// TIA Portal V16 export
// export: Created 2023-08-28T09:37:51.4907013Z, ExportSetting WithDefaults, DisplayName Totally Integrated Automation Portal, DisplayVersion V16 Update 6, DisplayName TIA Portal Version Control Interface, DisplayVersion V16 Update 2, DisplayName TIA Portal Openness, DisplayVersion V16 Update 6, DisplayName STEP 7 Professional, DisplayVersion V16 Update 6, DisplayName STEP 7 Safety, DisplayVersion V16, DisplayName WinCC Advanced, DisplayVersion V16 Update 6
DATA_BLOCK "dbModbusRTU_Reg"   // DB37
TITLE = Modbus RTU Data
{ S7_Optimized_Access := 'FALSE' }
AUTHOR : RTecmer
VERSION : 0.1
// Dane pomiarowe przekazane z bloku danych master modbus RTU
// stored: AutoNumber true, DBAccessibleFromOPCUA true, IsOnlyStoredInLoadMemory false, IsWriteProtectedInAS false
   VAR
      received_6_Wielkość_przeływu_Adres_0 { S7_SetPoint := 'True'} : "typeDataABB_DWord";   // wielkość przepływu
      received_6_Licznik_objętość_VF_Adres_2 { S7_SetPoint := 'True'} : "typeDataABB_DWord";   // licznik objętości VF
      received_6_Licznik_objętość_VR_Adres_4 { S7_SetPoint := 'True'} : "typeDataABB_DWord";   // licznik objętości VR
      received_6_Licznik_różnicowy_VD_Adres_6 { S7_SetPoint := 'True'} : "typeDataABB_DWord";   // licznik różnicy
      receive_6_Stan_licz_bjętości_GF_Adres_8 { S7_SetPoint := 'True'} : "typeDataABB_DWord";   // licznik objetosci GF
      received_6_Stan_licz_bjętości_GR_Adres_10 { S7_SetPoint := 'True'} : "typeDataABB_DWord";   // licznik objetości GR
      received_6_Stan_licz_rózicowego_obj_GD_Adres_12 { S7_SetPoint := 'True'} : "typeDataABB_DWord";   // licznik róznicowy
      received_6_Stan_urządzenia_1000 { S7_SetPoint := 'True'} : "typeDataInverter_Word";   // stan urządzenia
      received_ROL_aktualny_przeływu_Adres_0 { S7_SetPoint := 'True'} : "typeDataABB_DWord";   // wielkość przepływu
      received_ROL_suma_objętość_VF_Adres_2 { S7_SetPoint := 'True'} : "typeDataABB_DWord";   // licznik objętości VF
      received_ROL_suma_objętość_VR_Adres_4 { S7_SetPoint := 'True'} : "typeDataABB_DWord";   // licznik objętości VR
      received_ROL__VD_Adres_6 { S7_SetPoint := 'True'} : "typeDataABB_DWord";   // licznik różnicy
      received_ROL__GF_Adres_8 { S7_SetPoint := 'True'} : "typeDataABB_DWord";   // licznik objetosci GF
      received_ROL__10 { S7_SetPoint := 'True'} : "typeDataABB_DWord";   // licznik objetości GR
      received_ROL__GD_Adres_12 { S7_SetPoint := 'True'} : "typeDataABB_DWord";   // licznik róznicowy
      received_Data_Stan_urządzenia_1000 { S7_SetPoint := 'True'} : "typeDataInverter_Word";   // stan urządzenia
      receivede26_Inver_Control_word_416000 { S7_SetPoint := 'True'} : "typeDataInverter_Word";   // Sowo komtrolneCTW falownika [Uint16, index 0]
      received26_Inver_setpoint_ref_416020 { S7_SetPoint := 'True'} : "typeDataInverter_Word";   // Słowo wartość zadana Hz [Int16, index -1]
      received26_Inver_Status_word_416030 { S7_SetPoint := 'True'} : "typeDataInverter_Word";   // Słowo statusu STW falownika [Uint16, index 0]
      received26_Inver_Frequency_416130 { S7_SetPoint := 'True'} : "typeDataInverter_Word";   // Słowo częstotliwość na wyjściu [Uint16, index -1]
      received26_Inver_MotorCurrent_416140 { S7_SetPoint := 'True'} : "typeDataInverter_Word";   // Słowo prąd na wyjściu [Uint16, index -2]
      received26_Inver_DC_Voltage_416300 { S7_SetPoint := 'True'} : "typeDataInverter_Word";   // Słowo napięcia DC na szynie [Uint16, index 0]
      received26_Inver_Temp_416340 { S7_SetPoint := 'True'} : "typeDataInverter_Word";   // Słowo temperatura invertera [Uint8, index 0]
      received26_Inver_NomCurrent_416360 { S7_SetPoint := 'True'} : "typeDataInverter_Word";   // Słowo nominalna wartośc prądu falonika[Uint16, index -2]
      received26_Inver_MaxCurrent_416370 { S7_SetPoint := 'True'} : "typeDataInverter_Word";   // Słowo max prąd falownika [Uint16, index -2]
      received26_Inver_InDigit_416600 { S7_SetPoint := 'True'} : "typeDataInverter_Word";   // Słowo mampa wejść 18,19,27,33 [Uint16, index -0]
      received26_Inver_HourWork_415010 { S7_SetPoint := 'True'} : "typeDataInverter_DWord";   // Podwójne słowo czasu pracy falownika [Int32, index -0]
      received26_Inver_OverTemp_415040 { S7_SetPoint := 'True'} : "typeDataInverter_Word";   // Sowo statusu przekroczenie temperatury[Uint16, index 0]
      received26_Inver_OverVolts_415050 { S7_SetPoint := 'True'} : "typeDataInverter_Word";   // Sowo statusu przekroczenie napięcia[Uint16, index 0]
      "Przepływomierz nr1 pompownia" : Struct
         ID6_przeływu_VF_Adres_0 { S7_SetPoint := 'True'} : Real;
         ID6_objętość_VF_Adres_2 { S7_SetPoint := 'True'} : Real;
         "ID6_objętośc RF_Adres_4" { S7_SetPoint := 'True'} : Real;
         ID6_licznik_różnicowy_VD_Adres_6 { S7_SetPoint := 'True'} : Real;
         ID6_licznik_objętości_GF_Adres_8 { S7_SetPoint := 'True'} : Real;
         ID6_Licznik_objętości_GR_Adres_10 { S7_SetPoint := 'True'} : Real;
         ID6_Licznik_różnicowy_GD_Adres_12 { S7_SetPoint := 'True'} : Real;
         ID6_status_przepływomierza_Adres_1000 { S7_SetPoint := 'True'} : Word;
      END_STRUCT;
      "Przepływomierz nr2" : Struct
         received_6_przeływu_VF_Adres_0 { S7_SetPoint := 'True'} : Real;
         received_6_objętość_VF_Adres_2 { S7_SetPoint := 'True'} : Real;
         "received_6_objętośc RF_Adres_4" { S7_SetPoint := 'True'} : Real;
         received_6_licznik_różnicowy_VD_Adres_7 { S7_SetPoint := 'True'} : Real;
         received_6_licznik_objętości_GF_Adres_8 { S7_SetPoint := 'True'} : Real;
         received_6_Licznik_objętości_GR_Adres_10 { S7_SetPoint := 'True'} : Real;
         received_6_Licznik_różnicowy_GD_Adres_12 { S7_SetPoint := 'True'} : Real;
         received_6_status_przepływomierza_Adres_1000 { S7_SetPoint := 'True'} : Word;
      END_STRUCT;
   END_VAR
BEGIN
END_DATA_BLOCK
